{attribute 'GeneratedUsingTerminal: EK1100-0000-0018'}
{attribute addProperty BoxType "EK1100-0000-0018"}
{attribute addProperty Id "Beckhoff_ELXxxxxEK1122Beckhoff_ELXxxxxEK1122_3FD8C7C72A_0001_ELX1052_0000_0016ELX1052_6CC2DB6A8A_0002_ELX1054_0000_0016ELX1054_EF479B4E16A_0003_ELX1058_0000_0016ELX1058_7670813D28A_0004_ELX2002_0000_0016ELX2002_B02149405A_0005_ELX2008_0000_0016ELX2008_E2806B9511A_0006_ELX3152_0000_0016ELX3152_AA20D87B32A_0007_ELX3152_0000_0017ELX3152_AA20D87B32A_0008_ELX3152_0090_0016ELX3152_AA20D87B32A_0009_ELX3152_0090_0017ELX3152_AA20D87B32A_0010_ELX3158_0000_0016ELX3158_35AE532492A_0011_ELX3181_0000_0016ELX3181_05065F7B28A_0012_ELX3181_0000_0017ELX3181_05065F7B28A_0013_ELX3202_0000_0016ELX3202_28AA99ED30A_0014_ELX3202_0090_0016ELX3202_28AA99ED30A_0015_ELX3204_0000_0016ELX3204_49A0002648A_0016_ELX3204_0090_0016ELX3204_49A0002648A_0017_ELX3252_0000_0016ELX3252_7FD1684B26A_0018_ELX3312_0000_0016ELX3312_792163DD30A_0019_ELX3312_0090_0016ELX3312_792163DD30A_0020_ELX3314_0000_0016ELX3314_B654D23048A_0021_ELX3314_0090_0016ELX3314_B654D23048A_0022_ELX3351_0000_0016ELX3351_DF51302B26A_0023_ELX3351_0090_0016ELX3351_DF51302B26A_0024_ELX4154_0000_0016ELX4154_D2A7C9B719A_0025_ELX4181_0000_0016ELX4181_7041D8BB19A_0026_ELX4181_0000_0017ELX4181_7041D8BB19A_0027_ELX5151_0000_0016ELX5151_C163EA3C25A_0028_ELX5151_0090_0016ELX5151_C163EA3C25A_0030_ELX9410_0000_0016ELX9410_6BC01D146A_0031_ELX9410_0000_0017ELX9410_6BC01D146A_0032_ELX9410_0000_0018ELX9410_089FA8546A_0033_ELX9560_0000_0016ELX9560_883C11A36A_0034_ELX9560_0000_0017ELX9560_883C11A36A_0035_ELX9560_0000_0018ELX9560_F22EDCF26"}
{attribute addProperty CRC "3646376629"}
{attribute addProperty Size "879"}
TYPE Beckhoff_ELXxxxx_D9574AB5 EXTENDS EK1100_1FC0878B :
STRUCT
	{attribute addProperty Name "Beckhoff_ELXxxxxEK1122"}
	{attribute addProperty PreviousPort "Beckhoff ELXxxxx : B"}
	Beckhoff_ELXxxxxEK1122 : Beckhoff_ELXxxxxEK1122_3FD8C7C7;
	{attribute addProperty Name "A_0001_ELX1052_0000_0016"}
	{attribute addProperty PreviousPort "Beckhoff ELXxxxxEK1122 : C"}
	A_0001_ELX1052_0000_0016 : ELX1052_6CC2DB6A;
	{attribute addProperty Name "A_0002_ELX1054_0000_0016"}
	{attribute addProperty PreviousPort "A_0001(ELX1052-0000-0016) : B"}
	A_0002_ELX1054_0000_0016 : ELX1054_EF479B4E;
	{attribute addProperty Name "A_0003_ELX1058_0000_0016"}
	{attribute addProperty PreviousPort "A_0002(ELX1054-0000-0016) : B"}
	A_0003_ELX1058_0000_0016 : ELX1058_7670813D;
	{attribute addProperty Name "A_0004_ELX2002_0000_0016"}
	{attribute addProperty PreviousPort "A_0003(ELX1058-0000-0016) : B"}
	A_0004_ELX2002_0000_0016 : ELX2002_B0214940;
	{attribute addProperty Name "A_0005_ELX2008_0000_0016"}
	{attribute addProperty PreviousPort "A_0004(ELX2002-0000-0016) : B"}
	A_0005_ELX2008_0000_0016 : ELX2008_E2806B95;
	{attribute addProperty Name "A_0006_ELX3152_0000_0016"}
	{attribute addProperty PreviousPort "A_0005(ELX2008-0000-0016) : B"}
	A_0006_ELX3152_0000_0016 : ELX3152_AA20D87B;
	{attribute addProperty Name "A_0007_ELX3152_0000_0017"}
	{attribute addProperty PreviousPort "A_0006(ELX3152-0000-0016) : B"}
	A_0007_ELX3152_0000_0017 : ELX3152_AA20D87B;
	{attribute addProperty Name "A_0008_ELX3152_0090_0016"}
	{attribute addProperty PreviousPort "A_0007(ELX3152-0000-0017) : B"}
	A_0008_ELX3152_0090_0016 : ELX3152_AA20D87B;
	{attribute addProperty Name "A_0009_ELX3152_0090_0017"}
	{attribute addProperty PreviousPort "A_0008(ELX3152-0090-0016) : B"}
	A_0009_ELX3152_0090_0017 : ELX3152_AA20D87B;
	{attribute addProperty Name "A_0010_ELX3158_0000_0016"}
	{attribute addProperty PreviousPort "A_0009(ELX3152-0090-0017) : B"}
	A_0010_ELX3158_0000_0016 : ELX3158_35AE5324;
	{attribute addProperty Name "A_0011_ELX3181_0000_0016"}
	{attribute addProperty PreviousPort "A_0010(ELX3158-0000-0016) : B"}
	A_0011_ELX3181_0000_0016 : ELX3181_05065F7B;
	{attribute addProperty Name "A_0012_ELX3181_0000_0017"}
	{attribute addProperty PreviousPort "A_0011(ELX3181-0000-0016) : B"}
	A_0012_ELX3181_0000_0017 : ELX3181_05065F7B;
	{attribute addProperty Name "A_0013_ELX3202_0000_0016"}
	{attribute addProperty PreviousPort "A_0012(ELX3181-0000-0017) : B"}
	A_0013_ELX3202_0000_0016 : ELX3202_28AA99ED;
	{attribute addProperty Name "A_0014_ELX3202_0090_0016"}
	{attribute addProperty PreviousPort "A_0013(ELX3202-0000-0016) : B"}
	A_0014_ELX3202_0090_0016 : ELX3202_28AA99ED;
	{attribute addProperty Name "A_0015_ELX3204_0000_0016"}
	{attribute addProperty PreviousPort "A_0014(ELX3202-0090-0016) : B"}
	A_0015_ELX3204_0000_0016 : ELX3204_49A00026;
	{attribute addProperty Name "A_0016_ELX3204_0090_0016"}
	{attribute addProperty PreviousPort "A_0015(ELX3204-0000-0016) : B"}
	A_0016_ELX3204_0090_0016 : ELX3204_49A00026;
	{attribute addProperty Name "A_0017_ELX3252_0000_0016"}
	{attribute addProperty PreviousPort "A_0016(ELX3204-0090-0016) : B"}
	A_0017_ELX3252_0000_0016 : ELX3252_7FD1684B;
	{attribute addProperty Name "A_0018_ELX3312_0000_0016"}
	{attribute addProperty PreviousPort "A_0017(ELX3252-0000-0016) : B"}
	A_0018_ELX3312_0000_0016 : ELX3312_792163DD;
	{attribute addProperty Name "A_0019_ELX3312_0090_0016"}
	{attribute addProperty PreviousPort "A_0018(ELX3312-0000-0016) : B"}
	A_0019_ELX3312_0090_0016 : ELX3312_792163DD;
	{attribute addProperty Name "A_0020_ELX3314_0000_0016"}
	{attribute addProperty PreviousPort "A_0019(ELX3312-0090-0016) : B"}
	A_0020_ELX3314_0000_0016 : ELX3314_B654D230;
	{attribute addProperty Name "A_0021_ELX3314_0090_0016"}
	{attribute addProperty PreviousPort "A_0020(ELX3314-0000-0016) : B"}
	A_0021_ELX3314_0090_0016 : ELX3314_B654D230;
	{attribute addProperty Name "A_0022_ELX3351_0000_0016"}
	{attribute addProperty PreviousPort "A_0021(ELX3314-0090-0016) : B"}
	A_0022_ELX3351_0000_0016 : ELX3351_DF51302B;
	{attribute addProperty Name "A_0023_ELX3351_0090_0016"}
	{attribute addProperty PreviousPort "A_0022(ELX3351-0000-0016) : B"}
	A_0023_ELX3351_0090_0016 : ELX3351_DF51302B;
	{attribute addProperty Name "A_0024_ELX4154_0000_0016"}
	{attribute addProperty PreviousPort "A_0023(ELX3351-0090-0016) : B"}
	A_0024_ELX4154_0000_0016 : ELX4154_D2A7C9B7;
	{attribute addProperty Name "A_0025_ELX4181_0000_0016"}
	{attribute addProperty PreviousPort "A_0024(ELX4154-0000-0016) : B"}
	A_0025_ELX4181_0000_0016 : ELX4181_7041D8BB;
	{attribute addProperty Name "A_0026_ELX4181_0000_0017"}
	{attribute addProperty PreviousPort "A_0025(ELX4181-0000-0016) : B"}
	A_0026_ELX4181_0000_0017 : ELX4181_7041D8BB;
	{attribute addProperty Name "A_0027_ELX5151_0000_0016"}
	{attribute addProperty PreviousPort "A_0026(ELX4181-0000-0017) : B"}
	A_0027_ELX5151_0000_0016 : ELX5151_C163EA3C;
	{attribute addProperty Name "A_0028_ELX5151_0090_0016"}
	{attribute addProperty PreviousPort "A_0027(ELX5151-0000-0016) : B"}
	A_0028_ELX5151_0090_0016 : ELX5151_C163EA3C;
	{attribute addProperty Name "A_0030_ELX9410_0000_0016"}
	{attribute addProperty PreviousPort "A_0028(ELX5151-0090-0016) : B"}
	A_0030_ELX9410_0000_0016 : ELX9410_6BC01D14;
	{attribute addProperty Name "A_0031_ELX9410_0000_0017"}
	{attribute addProperty PreviousPort "A_0030(ELX9410-0000-0016) : B"}
	A_0031_ELX9410_0000_0017 : ELX9410_6BC01D14;
	{attribute addProperty Name "A_0032_ELX9410_0000_0018"}
	{attribute addProperty PreviousPort "A_0031(ELX9410-0000-0017) : B"}
	A_0032_ELX9410_0000_0018 : ELX9410_089FA854;
	{attribute addProperty Name "A_0033_ELX9560_0000_0016"}
	{attribute addProperty PreviousPort "A_0032(ELX9410-0000-0018) : B"}
	A_0033_ELX9560_0000_0016 : ELX9560_883C11A3;
	{attribute addProperty Name "A_0034_ELX9560_0000_0017"}
	{attribute addProperty PreviousPort "A_0033(ELX9560-0000-0016) : B"}
	A_0034_ELX9560_0000_0017 : ELX9560_883C11A3;
	{attribute addProperty Name "A_0035_ELX9560_0000_0018"}
	{attribute addProperty PreviousPort "A_0034(ELX9560-0000-0017) : B"}
	A_0035_ELX9560_0000_0018 : ELX9560_F22EDCF2;
END_STRUCT
END_TYPE
